(* PLC project Unnamed, Unknown Unnamed 1 *)
(* stored: creationDateTime 2025-10-24T15:23:11, modificationDateTime 2025-10-25T19:44:21 *)

PROGRAM program0
  VAR
    OutB AT %QX0.0 : BOOL := 0;  (* Output al LED de 7 Segmentos (b) *)
    Input1 AT %IX0.0 : BOOL := 0;  (* Input del Sensor de movimiento *)
    OutA AT %QX0.1 : BOOL := 0;  (* Output al LED de 7 Segmentos (a) *)
    OutF AT %QX0.2 : BOOL := 0;  (* Output al LED de 7 Segmentos (f) *)
    OutG AT %QX0.3 : BOOL := 0;  (* Output al LED de 7 Segmentos (g) *)
    OutC AT %QX0.4 : BOOL := 0;  (* Output al LED de 7 Segmentos (c) *)
    OutD AT %QX0.5 : BOOL := 0;  (* Output al LED de 7 Segmentos (d) *)
    OutE AT %QX0.6 : BOOL := 0;  (* Output al LED de 7 Segmentos (e) *)
  END_VAR
  VAR
    TRU : BOOL := 1;  (* Constante BOOL:TRUE *)
    TP0 : TP;  (* Pulsador TP; Tiempo de 5 seg *)
    TOF0 : TOF;  (* Off-Delay Timer (parte del pulsador) *)
    TP1 : TP;  (* Pulsador TP; Tiempo de 0.2 seg (parte del pulsador) *)
    TP2 : TP;  (* Pulsador TP; Tiempo de 3 seg *)
  END_VAR
  VAR  (* added by the conversion: wires and edge detectors of the diagram *)
    _AND15_OUT : BOOL;
    _OR27_OUT : BOOL;
  END_VAR

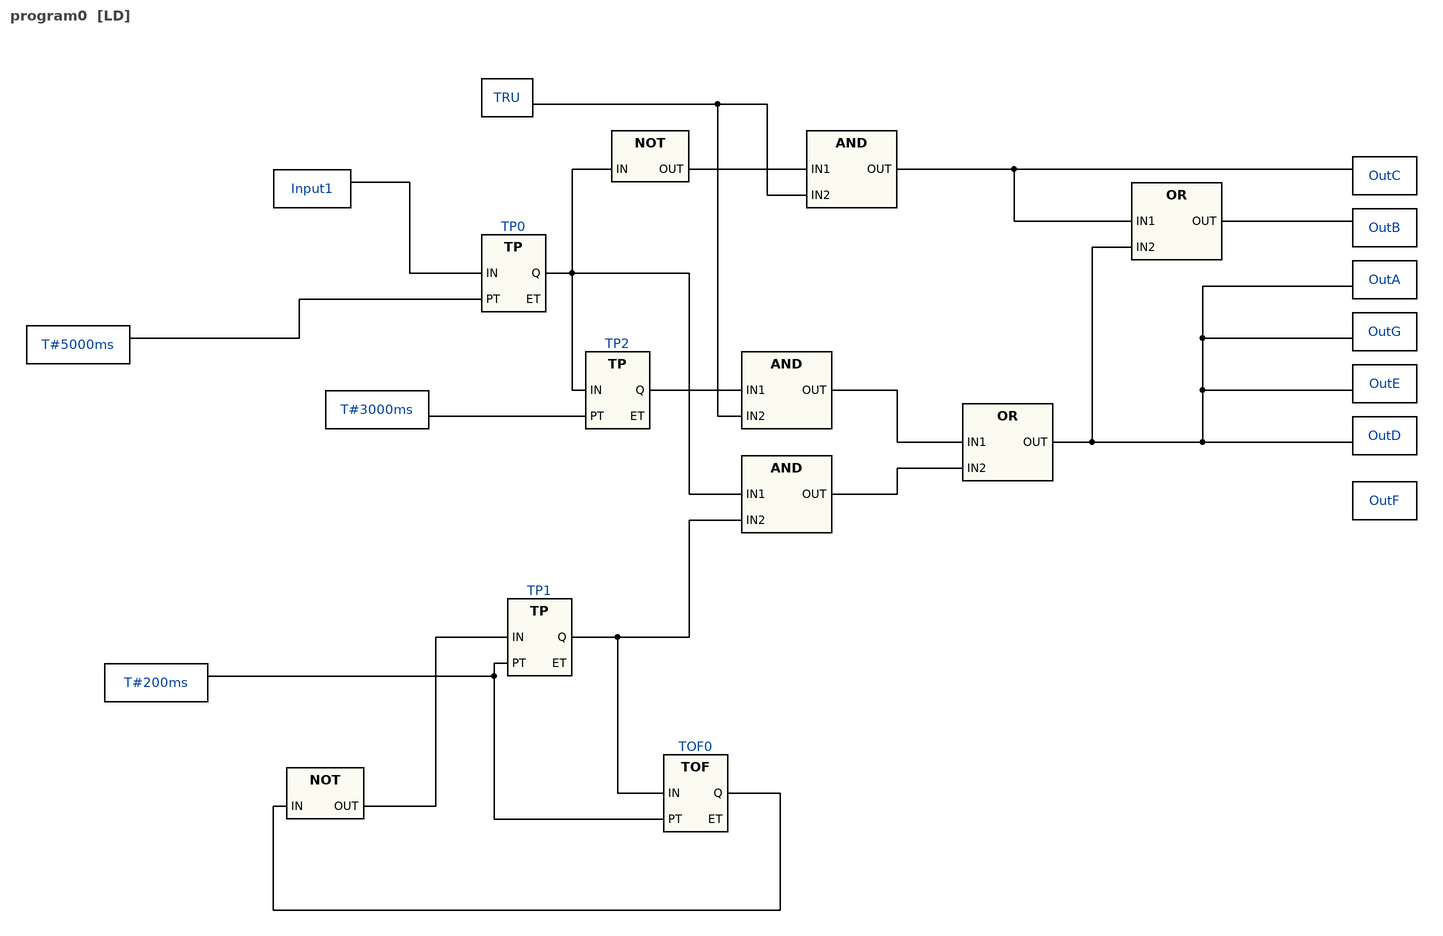
(* LD diagram, written out as Structured Text *)
TP0(IN := Input1, PT := T#5000ms);
_AND15_OUT := NOT TP0.Q AND TRU;
TP2(IN := TP0.Q, PT := T#3000ms);
TOF0(IN := TP1.Q, PT := T#200ms);
TP1(IN := NOT TOF0.Q, PT := T#200ms);
_OR27_OUT := TP2.Q AND TRU OR TP0.Q AND TP1.Q;
OutB := _AND15_OUT OR _OR27_OUT;
OutD := _OR27_OUT;
OutA := _OR27_OUT;
OutE := _OR27_OUT;
OutG := _OR27_OUT;
OutC := _AND15_OUT;
END_PROGRAM

CONFIGURATION Config0
  RESOURCE Res0 ON PLC
    TASK task0(INTERVAL := T#20ms, PRIORITY := 0);
    PROGRAM instance0 WITH task0 : program0;
  END_RESOURCE
END_CONFIGURATION
